{attribute 'conditionalshow'}
TYPE ST_UN_FLOAT_CONVERT_ULINT_LREAL :
UNION
	{attribute 'hide'}
	uliRawValue				: ULINT;					//Raw value as ulint
	{attribute 'hide'}
	lrValueFloat			: LREAL;					//Float value
END_UNION
END_TYPE

(* stored: Version 1.1.0.1, ProductVersion 3.1.4024.9
   DUT ST_UN_FLOAT_CONVERT_ULINT_LREAL: Id {29c0e84c-ec24-4969-91aa-8a7399a617ba} *)
